// TIA Portal project "Siemens_Python" (V15.1)
// Projeto para Comunicação entre Siemens e Python

(* hardware
DEVICE "S7-1200 station_1"  S7-1200 Station
   slot 0: "Rack_0"  S7-1200 Rack  Rack  V1.0
   slot 1: "PLC"  CPU 1211C DC/DC/DC  6ES7 211-1AE31-0XB0  V3.0
*)

// ===== PLC "PLC"  CPU 1211C DC/DC/DC =====

DATA_BLOCK "Data_Python"   // DB1
{ S7_Optimized_Access := 'FALSE' }
VERSION : 0.1
   VAR
      Bool1 : Bool;
      Bool2 : Bool;
      Bool3 : Bool;
      Bool4 : Bool;
      Bool5 : Bool;
      Bool6 : Bool;
   END_VAR
BEGIN
END_DATA_BLOCK

ORGANIZATION_BLOCK "Main"   // OB1, LAD, ProgramCycle
TITLE = "Main Program Sweep (Cycle)"
{ S7_Optimized_Access := 'TRUE' }
VERSION : 0.1
BEGIN
END_ORGANIZATION_BLOCK